(* IEC 61131-3 sources: simple-control-modules/src/Pusher, 4 files *)

(* ---- PusherStates.st ---- *)
NAMESPACE Simatic.Ax.SimpleControlModules
    TYPE
        PusherState : (Retracted, Pushing, Pushed, Retracting) := Retracted;
    END_TYPE
END_NAMESPACE

(* ---- IPusher.st ---- *)
NAMESPACE Simatic.Ax.SimpleControlModules
    INTERFACE IPusher
        METHOD Push END_METHOD
        METHOD Retract END_METHOD
        METHOD GetState : PusherState
        END_METHOD
    END_INTERFACE
END_NAMESPACE

(* ---- PusherBiDirTimeBased.st ---- *)
USING System.Timer;
USING Simatic.Ax.Io.Output;

NAMESPACE Simatic.Ax.SimpleControlModules
    CLASS PusherBiDirTimeBased IMPLEMENTS IPusher

        VAR PUBLIC
            ControlPush : IBinOutput;
            ControlRetract : IBinOutput;
            OnDuration : TIME;
            OffDuration : TIME;
            AutoRetract : BOOL := TRUE;
        END_VAR
        VAR
            _tonOnDuration : OnDelay;
            _tonOffDuration : OnDelay;
            _state : PusherState;
        END_VAR

        METHOD PUBLIC Evaluate
            _tonOnDuration(signal := _state = PusherState#Pushing);
            _tonOffDuration(signal := _state = PusherState#Retracting);

            CASE _state OF
                PusherState#Retracted :
                    ControlRetract.SetOff();

                PusherState#Pushing :
                    ControlPush.SetOn();
                    IF (_tonOnDuration.output) THEN
                        _state := PusherState#Pushed;
                    END_IF;

                PusherState#Pushed :
                    ControlPush.SetOff();
                    IF (AutoRetract) THEN
                        _state := PusherState#Retracting;
                    END_IF;

                PusherState#Retracting :
                    ControlRetract.SetOn();
                    IF (_tonOffDuration.output) THEN
                        _state := PusherState#Retracted;
                    END_IF;
            END_CASE;

        END_METHOD

        METHOD PUBLIC Push
            IF (_state = PusherState#Retracted OR _state = PusherState#Retracting) THEN
                _state := PusherState#Pushing;
                _tonOnDuration.duration := OnDuration;
            END_IF;
        END_METHOD

        METHOD PUBLIC Retract
            _state := PusherState#Retracting;
        END_METHOD

        METHOD PUBLIC GetState : PusherState
            GetState := _state;
        END_METHOD
    END_CLASS
END_NAMESPACE

(* ---- PusherTimeBased.st ---- *)
USING System.Timer;
USING Simatic.Ax.Io.Output;

NAMESPACE Simatic.Ax.SimpleControlModules
    CLASS PusherTimeBased IMPLEMENTS IPusher

        VAR PUBLIC
            ControlPush : IBinOutput;
            OnDuration : TIME;
        END_VAR
        VAR
            _tonOnDuration : OnDelay;
            _state : PusherState;
        END_VAR

        METHOD PUBLIC Evaluate
            _tonOnDuration(signal := _state = PusherState#Pushing);

            CASE _state OF
                PusherState#Retracted :
                    ControlPush.SetOff();

                PusherState#Pushing :
                    ControlPush.SetOn();
                    IF (_tonOnDuration.output) THEN
                        _state := PusherState#Retracting;
                        ControlPush.SetOff();
                    END_IF;

                PusherState#Retracting :
                    ControlPush.SetOff();
                    _state := PusherState#Retracted;
            END_CASE;

        END_METHOD

        METHOD PUBLIC Push
            _state := PusherState#Pushing;
        END_METHOD

        METHOD PUBLIC Retract
            _state := PusherState#Retracted;
        END_METHOD

        METHOD PUBLIC GetState : PusherState
            GetState := _state;
        END_METHOD
    END_CLASS
END_NAMESPACE
